// Mitsubishi GX Works2 project: EX2809SETRESET   PLC: Q03UDV

PROGRAM MAIN
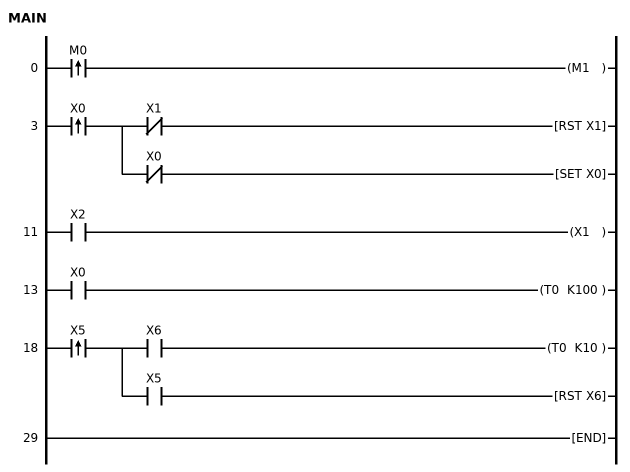
0     LDP     M0
      OUT     M1
3     LDP     X0
      MPS
      ANI     X1
      RST     X1
      MPP
      ANI     X0
      SET     X0
11    LD      X2
      OUT     X1
13    LD      X0
      OUT     T0 K100
18    LDP     X5
      MPS
      AND     X6
      OUT     T0 K10
      MPP
      AND     X5
      RST     X6
29    END
END_PROGRAM
